FUNCTION_BLOCK FINAL Trigger
VAR_INPUT
END_VAR
VAR_OUTPUT
END_VAR
VAR
	rTrig : R_TRIG ;
	ftrig : F_TRIG ;
END_VAR

METHOD PUBLIC EDGENEG : BOOL
VAR_INPUT
	input : BOOL ;
END_VAR

fTrig.CLK := input ;
fTrig();

EDGENEG := fTrig.Q ;
END_METHOD

METHOD PUBLIC EDGEPOS : BOOL
VAR_INPUT
	input : BOOL ;
END_VAR

rTrig.CLK := input ;
rTrig();

EDGEPOS := rTrig.Q ;
END_METHOD

METHOD ONE_SHOT : BOOL
VAR_INPUT
	input : BOOL ;
END_VAR
rTrig.CLK := input ;
rTrig();

fTrig.CLK := input ;
fTrig();

ONE_SHOT := rTrig.Q OR fTrig.Q;
END_METHOD

END_FUNCTION_BLOCK

(* stored: Version 1.1.0.1, ProductVersion 3.1.4024.3
   POU Trigger: Id {c67d9166-d540-0202-2a88-8baffae3daa6}, SpecialFunc None
   Method EDGENEG: Id {8b9bf463-f22b-095e-1db4-d63fc4c7cc31}
   Method EDGEPOS: Id {1b4843c4-926f-0a87-1a67-26986fba09a2}
   Method ONE_SHOT: Id {fa5bf7b6-b5ec-0068-3543-831b1fbdbce5} *)
